FUNCTION_BLOCK FB_Recipes
VAR_INPUT
	xICreateRecipe:BOOL;
	xILoadRecipe:BOOL;
	xIDeleteRecipe:BOOL;
	strRecipeDefinitionName:STRING:='Recipes';
	RecipeName:STRING:='';
	FileName: STRING (255):='';
	
END_VAR
VAR_OUTPUT
END_VAR
VAR
	fbRecipeManCommands:Recipe_Management.RecipeManCommands;
	dwReturnCreate:DWORD;
	dwReturnWrite:DWORD;
	dwReturnRead:DWORD;
	dwReturnDelete:DWORD;
	dwSetPath		:DWORD;
	dwReturnDeleteFile: DWORD;
	xRecipeCreate:BOOL;
	xRecipeDelete:BOOL;
	xRecipeRead:BOOL;
	xRecipeWrite:BOOL;
	xLoadRecipe:BOOL;
	xSetPath:BOOL;
	
	
	stPath:STRING:='\Hard Disk1\prog\';//CE系统路径
	wActionStep:WORD;
	wActionStep1: WORD;
	wActionStep2: WORD;
	
	dwReturnLoadFromAndWrite: DWORD;
	
	dwResetLastError: DWORD;
END_VAR
VAR_OUTPUT
	xQBusy:BOOL;
	xQErrorID:DWORD;
END_VAR

VAR CONSTANT
	ERR_OK                                     	:DWORD:=16#0000;//Result OK
	ERR_NO_RECIPE_MANAGER_SET                 	:DWORD:=16#4006;//The global recipe manager has not been created.
	ERR_RECIPE_DEFINITION_NOT_FOUND           	:DWORD:=16#4004;  //The recipe definition does not exist.                                      
	ERR_RECIPE_ALREADY_EXIST                  	:DWORD:=16#4005; //The recipe already exists in the recipe definition. Create a new recipe under a different name                                     
	ERR_RECIPE_NOMEMORY                       	:DWORD:=16#4008;  //  The recipe definition has no free memory to create a new recipe.                        
	ERR_RECIPE_NOT_FOUND                        :DWORD:=16#4003; //The recipe does not exist                                          
	ERR_RECIPE_FILE_NOT_FOUND                   :DWORD:=16#4000;//The recipe file was not found.
END_VAR

ACT_Create();
ACT_Delete();
ACT_Read();
IF   wActionStep =0 AND   wActionStep1 =0  AND wActionStep2=0 THEN
	xQBusy:=FALSE;
ELSE
	xQBusy:=TRUE;
END_IF
IF  xQErrorID<>ERR_OK THEN
	dwResetLastError:=fbRecipeManCommands.ResetLastError();
			
END_IF

ACTION ACT_Create:
CASE wActionStep OF
	0:
		IF  xICreateRecipe THEN
			xICreateRecipe:=FALSE;
			wActionStep:=10;
			
		END_IF
	10: //创建配方保存路径
	 	xSetPath:=fbRecipeManCommands.SetStoragePath(stPath:=(*stPath*)'\Hard Disk1\Recipefiles\' );
		wActionStep:=20;
	20:	
		IF   xSetPath THEN
		
			wActionStep:=30;
		END_IF
	30:  ///(*创建一个配方，并且把当前PLC数据写入到配方中*)
		dwReturnCreate:=fbRecipeManCommands.CreateRecipe(RecipeDefinitionName:=strRecipeDefinitionName , RecipeName:=RecipeName );
		wActionStep:=40;
	40: 
		IF  dwReturnCreate =ERR_OK  OR    dwReturnCreate =ERR_RECIPE_ALREADY_EXIST  THEN
			
			wActionStep:=50;
		ELSE
			xQErrorID:=dwReturnCreate;
		END_IF
	50:  //将PLC数据写入到配方中去
			dwReturnRead:=fbRecipeManCommands.ReadRecipe(RecipeDefinitionName:= strRecipeDefinitionName, RecipeName:=RecipeName );
			wActionStep:=60;
	60:
		 IF   dwReturnRead =ERR_OK THEN
			
			 wActionStep:=70;
		ELSE
			xQErrorID:=dwReturnRead;
		 END_IF
	70:   	
			wActionStep:=0;
END_CASE
END_ACTION

ACTION ACT_Delete:

CASE wActionStep2 OF
	0:
		IF  xILoadRecipe THEN
			xILoadRecipe:=FALSE;
			wActionStep2:=10;
		END_IF
	10: //删除配方
	 	dwReturnDelete:=fbRecipeManCommands.DeleteRecipe(RecipeDefinitionName:=strRecipeDefinitionName , RecipeName:=RecipeName );
		wActionStep2:=20;
	20:	
		IF   dwReturnDelete= ERR_OK THEN
			wActionStep2:=30;
		ELSE
			xQErrorID:=dwReturnDelete;
		END_IF
	30://删除配方文件
		dwReturnDeleteFile:=fbRecipeManCommands.DeleteRecipeFile(RecipeDefinitionName:= strRecipeDefinitionName , RecipeName:=RecipeName );
		wActionStep2:=40;	
	40:		
		IF   dwReturnDeleteFile= ERR_OK THEN
			wActionStep2:=50;
		ELSE
			xQErrorID:=dwReturnDeleteFile;
		END_IF
	50:   wActionStep2:=0;
END_CASE
END_ACTION

ACTION ACT_Read:

CASE wActionStep1 OF
	0:
		IF  xILoadRecipe THEN
			xILoadRecipe:=FALSE;
			wActionStep1:=10;
		END_IF
		
	
	10: //读取配方数据，写入PLC变量中
	 		dwReturnRead:=fbRecipeManCommands.ReadAndSaveRecipe(RecipeDefinitionName:= strRecipeDefinitionName, RecipeName:=RecipeName );
		(*dwReturnLoadFromAndWrite:=fbRecipeManCommands.LoadFromAndWriteRecipe(RecipeDefinitionName:=strRecipeDefinitionName , RecipeName:=RecipeName , FileName:=FileName );*)
		(*dwReturnWrite:=fbRecipeManCommands.WriteRecipe(RecipeDefinitionName:= strRecipeDefinitionName, RecipeName:=RecipeName );*)
		(*dwReturnLoadFromAndWrite:=fbRecipeManCommands.ReadRecipe(RecipeDefinitionName:=strRecipeDefinitionName , RecipeName:=RecipeName );*)
		IF  dwReturnRead>0 THEN
			wActionStep1:=20;
		END_IF
	20:	
		IF   dwReturnLoadFromAndWrite= ERR_OK THEN
			wActionStep1:=30;
		ELSE
			xQErrorID:=dwReturnLoadFromAndWrite;
		END_IF
	30:   wActionStep1:=0;
END_CASE
END_ACTION

END_FUNCTION_BLOCK

(* stored: Version 1.1.0.1, ProductVersion 3.1.4024.9
   POU FB_Recipes: Id {850c5608-11a9-488d-9dba-0d4d2e0cbc10}, SpecialFunc None
   Action ACT_Create: Id {d7eaaf49-7b9e-457e-9557-df95981b2860}
   Action ACT_Delete: Id {7f98c8e3-f269-4fef-8331-b86c9c8ddc00}
   Action ACT_Read: Id {7a2c162f-48f9-4cec-93fb-b3762e117bdf} *)
